// TIA Portal V17 export
// export: Created 2023-05-07T12:12:21.9941394Z, ExportSetting WithDefaults, DisplayName Totally Integrated Automation Portal, DisplayVersion V17, DisplayName TIA Portal Openness, DisplayVersion V17, DisplayName TIA Portal Version Control Interface, DisplayVersion V17, DisplayName TIA Portal Test Suite Advanced, DisplayVersion V17, DisplayName STEP 7 Professional, DisplayVersion V17, DisplayName SIMATIC Energy Suite, DisplayVersion V17, DisplayName STEP 7 Safety, DisplayVersion V17, DisplayName WinCC Professional, DisplayVersion V17
DATA_BLOCK "VisuData"   // DB9
{ S7_Optimized_Access := 'TRUE' }
VERSION : 0.1
// stored: AutoNumber true, IsOnlyStoredInLoadMemory false, IsRetainMemResEnabled false, IsWriteProtectedInAS false, MemoryReserve 100
   VAR
      Start : Bool;
      Stop : Bool;
      Empty : Bool;
      Controller : Int;
      RandomDisturbance : Int;
      SetPoint : Real;
      Outflow : Real;
      LevelMeterShow : Real;
      SetPointShow : Real;
      FillValveShow : Real;
      TopPump : Int;
      LowPump : Int;
      Status : Bool;
      default : Bool;
      finish_training : Int;
      factoryio_connect : Bool;
   END_VAR
BEGIN
END_DATA_BLOCK
